(* Logix 5000 project; controller blank vendor 1 type 14 code 96 rev 28.11; software revision 28.00 *)

TASK MainTask (continuous, watchdog 500 ms) : MainProgram

MODULES
   Local : vendor 1 type 14 code 96 (ICP 1, rev 28.11)
      relay_output_2 : 1756-IB16 (ICP 2, rev 3.4, Input RPI 20 ms)
      relay_output_4 : 1756-OW16I (ICP 4, rev 3.1, Output RPI 20 ms)
      realy_output_0 : 1756-OW16I (ICP 0, rev 3.1, Output RPI 20 ms)
      relay_output_8 : 1756-IF6I (ICP 8, rev 1.1, Input RPI 100 ms)
      relay_output_7 : vendor 1 type 10 code 4 (ICP 7, rev 1.1, Output RPI 25 ms)
      relay_output_9 : vendor 1 type 12 code 219 (ICP 9, rev 10.1)
         DNET : 1734-AENTR (Ethernet 192.168.1.10, rev 5.1, Output RPI 20 ms)
            Input : vendor 1 type 7 code 307 (PointIO 1, rev 3.1)
            Input2 : vendor 1 type 7 code 307 (PointIO 3, rev 3.1)
            Input3 : vendor 1 type 7 code 307 (PointIO 4, rev 3.1)
            Input1 : vendor 1 type 7 code 307 (PointIO 2, rev 3.1)
            Output : vendor 1 type 7 code 134 (PointIO 5, rev 3.1)
            Output1 : vendor 1 type 7 code 134 (PointIO 6, rev 3.1)
            Output2 : vendor 1 type 7 code 134 (PointIO 7, rev 3.1)
END_MODULES

PROGRAM MainProgram   (* main routine MainRoutine *)
VAR
   RED_LIGHT : ALIAS FOR DNET:5:O.1;
   TIMER_1 : TIMER := (PRE := 10000);
   YELL : ALIAS FOR DNET:6:O.1;
END_VAR

ROUTINE MainRoutine   (* ladder *)
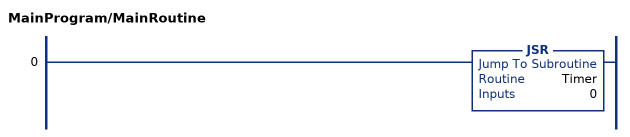
   0: JSR(Timer,0);
END_ROUTINE

ROUTINE Timer   (* ladder *)
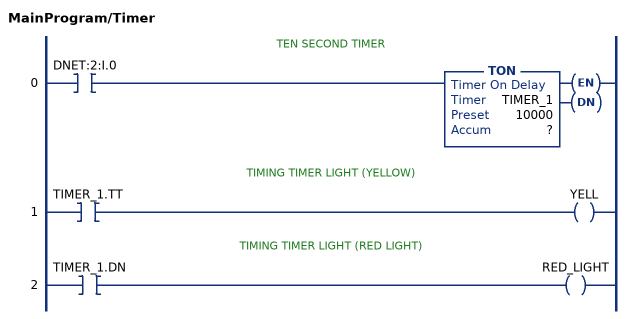
   // TEN SECOND TIMER
   0: XIC(DNET:2:I.0)TON(TIMER_1,?,?);
   // TIMING TIMER LIGHT (YELLOW)
   1: XIC(TIMER_1.TT)OTE(YELL);
   // TIMING TIMER LIGHT (RED LIGHT)
   2: XIC(TIMER_1.DN)OTE(RED_LIGHT);
END_ROUTINE
END_PROGRAM
